% RSLogix 500 project LAB3_BAK001.RSS, saved by version 8.30.00.16 %
PROJECT "LAB3"    % processor: Bul.1763 MicroLogix 1100 Series B %

PROGRAM FILES
  LAD 2   2 rungs

DATA FILES
  O0 OUTPUT  4 elements
  I1 INPUT  6 elements
  S2 STATUS  66 elements
  B3 BINARY  1 elements
  T4 TIMER  1 elements
  C5 COUNTER  1 elements
  R6 CONTROL  1 elements
  N7 INTEGER  1 elements
  F8 FLOAT  1 elements

LADDER 2
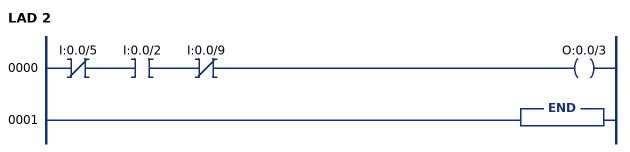
% Rung: 0 %
SOR XIO I:0.0/5 XIC I:0.0/2 XIO I:0.0/9 OTE O:0.0/3 EOR
% Rung: 1 %
SOR END EOR
